Universal Robots PolyScope program: ExtendTest.urp

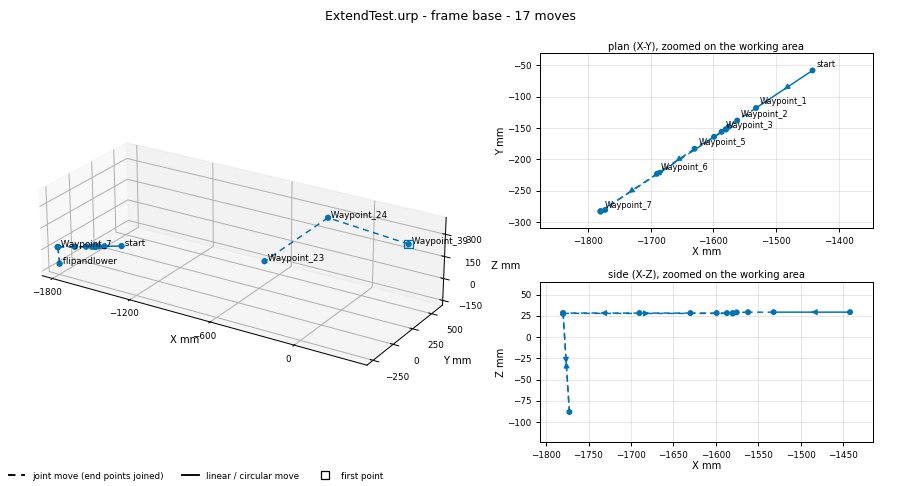
[picture p0: tool path of ExtendTest.urp in frame base, 17 of 19 moves have a stored position in this frame; points joined in program order, loops and branches not executed]
Program ExtendTest (installation=default directory=/programs createdIn=5.14.5 lastSavedIn=5.14.5 robotSerialNumber=20236801216)
Calibrated DH parameters: a=[-0.000021, -0.748897, -0.28186, -0.00004, -0.000055, 0]; d=[0.236225, -424.082933, -1564.66872, 1988.95162, 0.159094, 0.153873]; alpha=[1.570844, 0.001002, 0.000337, 1.571488, -1.569996, 0]; deltaTheta=[0, -0.516316, 5.626292, 1.173211, 0.000001, 0]
InitVariablesNode
Robot Program (runOnlyOnce=true)
  Script file /programs/usbdisk/robotTestScript.script
    | p_5 = p[-1.4420008419286459, -0.058094127721509764, 0.029525, -1.6440472482117785, 0.8546511027915219, 1.6440472482117785]
    | p_4 = p[-1.1727715142479016, 0.1308781295454616, 0.029525, -1.6440472482117785, 0.8546511027915219, 1.6440472482117785]
  p_4 := p_4
  p_5 := p_5
  SafeHome (positionOptionType=SPEED_AND_ACCELERATION speed=1.047198 acceleration=1.396263 nextMotionTime=2)
  MoveJ speed 60 deg/s, acceleration 80 deg/s^2 (useActiveTCP=true) feature=Base
    Waypoint Waypoint_39: TCP in base x=397.377 y=356.253 z=319.81 mm, rx=2.3163 ry=2.0576 rz=0.0741 rad; joints [-198.126, -117.851, 133.304, -13.01, -11.422, -6.036] deg; TCP offset x=-5.49 y=-328 z=106.39 mm, rx=1.2092 ry=-1.2092 rz=1.2092 rad
    Waypoint Waypoint_24: TCP in base x=-308.526 y=606.096 z=242.373 mm, rx=-2.1337 ry=0.3494 rz=2.1309 rad; joints [-107.196, -73.784, 125.643, 43.029, 90.975, 86.468] deg; TCP offset x=-4.211 y=-279.829 z=105.916 mm, rx=1.2092 ry=-1.2092 rz=1.2092 rad
  MoveJ speed 60 deg/s, acceleration 80 deg/s^2 (useActiveTCP=true) feature=Base
    Waypoint Waypoint_23: TCP in base x=-540.167 y=215.949 z=34.631 mm, rx=-1.5058 ry=1.0576 rz=1.5735 rad; joints [-26.452, -65.119, 143.749, 8.723, 85.674, 218.843] deg
  MoveJ speed 60 deg/s, acceleration 80 deg/s^2 (useActiveTCP=true) feature=Base
    Waypoint Variable (Variable): variable=p_4
  MoveL speed 12 mm/s, acceleration 1200 mm/s^2 (useActiveTCP=true) feature=Base
    Waypoint Variable (Variable): variable=p_5
  MoveJ speed 60 deg/s, acceleration 80 deg/s^2 (useActiveTCP=true) feature=Base
    Waypoint start: TCP in base x=-1441.999 y=-58.08 z=29.501 mm, rx=-1.6441 ry=0.8547 rz=1.644 rad; joints [5.647, -25.42, 51.127, 64.248, 89.949, 240.561] deg; TCP offset x=-5.49 y=-328 z=106.39 mm, rx=1.2092 ry=-1.2092 rz=1.2092 rad
  MoveL speed 250 mm/s, acceleration 1200 mm/s^2 (useActiveTCP=true) feature=Base
    Waypoint Waypoint_1: TCP in base x=-1531.999 y=-117.968 z=29.479 mm, rx=-1.6441 ry=0.8546 rz=1.644 rad; joints [7.758, -15.327, 29.134, 76.151, 89.944, 242.678] deg
  MoveJ speed 60 deg/s, acceleration 80 deg/s^2 (useActiveTCP=true) feature=Base
    Waypoint Waypoint_2: TCP in base x=-1562.007 y=-137.918 z=29.457 mm, rx=-1.6441 ry=0.8546 rz=1.6439 rad; joints [8.392, -9.44, 16.333, 83.066, 89.942, 243.317] deg
  MoveJ speed 60 deg/s, acceleration 80 deg/s^2 (useActiveTCP=true) feature=Base
    Waypoint degree1elbow: TCP in base x=-1575.447 y=-147.751 z=29.231 mm, rx=-1.6441 ry=0.8546 rz=1.6438 rad; joints [8.699, -2.629, 1.516, 91.078, 89.941, 243.632] deg
  MoveJ speed 60 deg/s, acceleration 80 deg/s^2 (useActiveTCP=true) feature=Base
    Waypoint afterspin: TCP in base x=-1580.228 y=-152.119 z=28.324 mm, rx=-1.6456 ry=0.8568 rz=1.6399 rad; joints [8.799, 30.631, -73.231, -47.231, -89.817, 63.802] deg
  MoveJ speed 60 deg/s, acceleration 80 deg/s^2 (useActiveTCP=true) feature=Base
    Waypoint Waypoint_3: TCP in base x=-1586.993 y=-155.992 z=28.382 mm, rx=-1.6455 ry=0.8568 rz=1.6398 rad; joints [8.91, 30.233, -72.29, -47.775, -89.815, 63.915] deg
  MoveJ speed 60 deg/s, acceleration 80 deg/s^2 (useActiveTCP=true) feature=Base
    Waypoint Waypoint_4: TCP in base x=-1599.002 y=-163.994 z=28.431 mm, rx=-1.6455 ry=0.8568 rz=1.6399 rad; joints [9.149, 29.5, -70.555, -48.779, -89.814, 64.151] deg
  MoveJ speed 60 deg/s, acceleration 80 deg/s^2 (useActiveTCP=true) feature=Base
    Waypoint Waypoint_5: TCP in base x=-1630 y=-182.994 z=28.402 mm, rx=-1.6456 ry=0.8568 rz=1.6398 rad; joints [9.681, 27.542, -65.949, -51.426, -89.812, 64.682] deg
  MoveJ speed 60 deg/s, acceleration 80 deg/s^2 (useActiveTCP=true) feature=Base
    Waypoint Waypoint_6: TCP in base x=-1689.998 y=-222.977 z=28.391 mm, rx=-1.6456 ry=0.8568 rz=1.6398 rad; joints [10.762, 23.212, -55.93, -57.117, -89.807, 65.759] deg
  MoveJ speed 60 deg/s, acceleration 80 deg/s^2 (useActiveTCP=true) feature=Base
    Waypoint Waypoint_7: TCP in base x=-1779.999 y=-282.991 z=28.44 mm, rx=-1.6455 ry=0.8568 rz=1.6399 rad; joints [12.221, 14.58, -36.424, -67.997, -89.804, 67.21] deg
  MoveJ speed 60 deg/s, acceleration 80 deg/s^2 (useActiveTCP=true) feature=Base
    Waypoint flipandlower: TCP in base x=-1772.528 y=-280.496 z=-88.099 mm, rx=-1.6606 ry=0.837 rz=1.6133 rad; joints [12.221, -14.579, 36.42, -110, -89.803, 67.209] deg
  MoveJ speed 60 deg/s, acceleration 80 deg/s^2 (useActiveTCP=true) feature=Base
    Waypoint flipped: TCP in base x=-1779.842 y=-282.887 z=27.59 mm, rx=-1.6608 ry=0.8367 rz=1.6129 rad; joints [12.248, -18.08, 34.479, -104.536, -89.806, 67.235] deg
  MoveJ speed 60 deg/s, acceleration 80 deg/s^2 (useActiveTCP=true) feature=Base
    Waypoint flippedexact: TCP in base x=-1780.087 y=-282.746 z=28.051 mm, rx=-1.6458 ry=0.8569 rz=1.64 rad; joints [12.238, -18.68, 36.443, -107.608, -89.796, 67.19] deg
  MoveJ speed 60 deg/s, acceleration 80 deg/s^2 (useActiveTCP=true) feature=Base
    Waypoint Waypoint_8: TCP in base x=-1580.004 y=-152.009 z=27.98 mm, rx=-1.6459 ry=0.8568 rz=1.64 rad; joints [8.846, -35.474, 73.269, -127.627, -89.813, 63.792] deg
